Omron Sysmac Studio project AccumulationTimer_TP_Timer (Sysmac Studio 1.65.0.64007, StandardProject)

# Controller new_Controller_0: NX1P2-1040DT1 version 1.69
Task PrimaryTask (priority 4, period or condition 2000): Program0

VAR_GLOBAL
    BIO_Input_Bit_00 : BOOL;  (* at BuiltInIO://cpu/#0/Input_Bit_00 *)
    BIO_Input_Bit_01 : BOOL;  (* at BuiltInIO://cpu/#0/Input_Bit_01 *)
    BIO_Output_Bit_00 : BOOL;  (* at BuiltInIO://cpu/#0/Output_Bit_00 *)
    BIO_Output_Bit_01 : BOOL;  (* at BuiltInIO://cpu/#0/Output_Bit_01 *)
    IN_Start_Button : BOOL;
    INP : BOOL;
    StartButton : BOOL;
    StopButton : BOOL;
    Motor1 : BOOL;
    Motor2 : BOOL;
    AccumTimer1_Reset : BOOL;
    AccumTimer1_ET : TIME;
    Motor1_CalismaSuresi : INT;
    OUT_Motor1_Start : BOOL;
    OUT_Motor2_Start : BOOL;
    AccumTimer2_Reset : BOOL;
    AccumTimer2_ET : TIME;
    Motor2_CalismaSuresi : INT;
END_VAR

PROGRAM Program0
VAR
    Start : BOOL;
    AccumTimer1 : AccumulationTimer;
    AccumTimer2 : AccumulationTimer;
END_VAR
VAR_EXTERNAL
    IN_Start_Button : BOOL;
    BIO_Output_Bit_00 : BOOL;
    INP : BOOL;
    BIO_Input_Bit_00 : BOOL;
    StartButton : BOOL;
    BIO_Input_Bit_01 : BOOL;
    StopButton : BOOL;
    Motor1 : BOOL;
    Motor2 : BOOL;
    BIO_Output_Bit_01 : BOOL;
    AccumTimer1_Reset : BOOL;
    AccumTimer1_ET : TIME;
    Motor1_CalismaSuresi : INT;
    OUT_Motor1_Start : BOOL;
    OUT_Motor2_Start : BOOL;
    AccumTimer2_Reset : BOOL;
    AccumTimer2_ET : TIME;
    Motor2_CalismaSuresi : INT;
END_VAR
VAR
    _e1 : R_TRIG;
    _e2 : R_TRIG;
END_VAR

(* Section InOut: ladder, written here as Structured Text *)

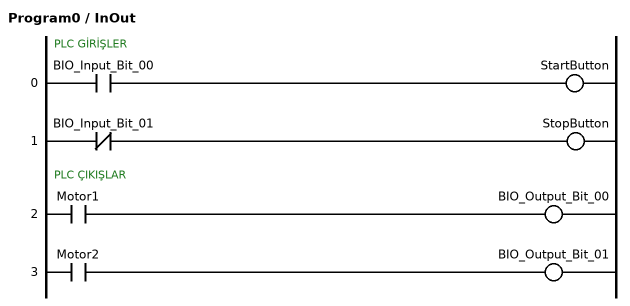
(* Rung 0: PLC GİRİŞLER *)
StartButton := BIO_Input_Bit_00;
(* Rung 1 *)
StopButton := NOT BIO_Input_Bit_01;
(* Rung 2: PLC ÇIKIŞLAR *)
BIO_Output_Bit_00 := Motor1;
(* Rung 3 *)
BIO_Output_Bit_01 := Motor2;

(* Section Timerr: ladder, written here as Structured Text *)

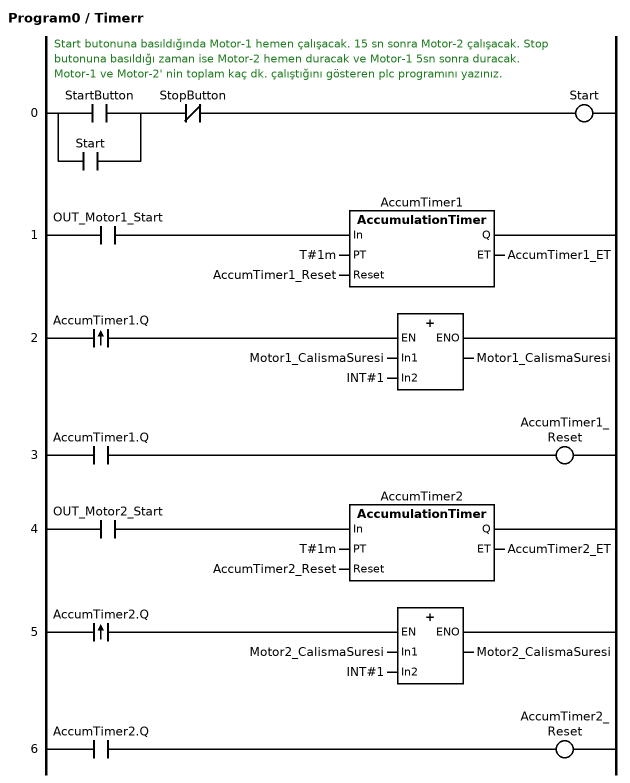
(* Rung 0: Start butonuna basıldığında Motor-1 hemen çalışacak. 15 sn sonra Motor-2 çalışacak. Stop butonuna basıldığı zaman ise Motor-2 hemen duracak ve Motor-1 5sn sonra duracak. Motor-1 ve Motor-2' nin toplam kaç dk. çalıştığını gösteren plc programını yazınız. *)
Start := (StartButton OR Start) AND NOT StopButton;
(* Rung 1 *)
AccumTimer1(In := OUT_Motor1_Start, PT := T#1m, Reset := AccumTimer1_Reset, ET => AccumTimer1_ET);
(* Rung 2 *)
_e1(CLK := AccumTimer1.Q);
IF _e1.Q THEN Motor1_CalismaSuresi := Motor1_CalismaSuresi + INT#1; END_IF;
(* Rung 3 *)
AccumTimer1_Reset := AccumTimer1.Q;
(* Rung 4 *)
AccumTimer2(In := OUT_Motor2_Start, PT := T#1m, Reset := AccumTimer2_Reset, ET => AccumTimer2_ET);
(* Rung 5 *)
_e2(CLK := AccumTimer2.Q);
IF _e2.Q THEN Motor2_CalismaSuresi := Motor2_CalismaSuresi + INT#1; END_IF;
(* Rung 6 *)
AccumTimer2_Reset := AccumTimer2.Q;
END_PROGRAM